/// This the main class of the library. It represents a Pushover app and
/// is tied to a unique API token. When constructing the object it is mandatory to pass
/// an `app-token` as well as a `user-token`.
///
/// Here's a simple example, which sends a pushover notification to a specific device of the user.
/// Note that this class uses a fluent API to configure the properties of a notification.
/// The actual action of sending the notification is triggered by [SendMessageAsync](xref:Pushover.PushoverClient#SendMessageAsync).
/// The ´Async´ Suffix in this method indicates that this action has to be waited for by checking for ´NOT _pushoverClient.Busy´ before
/// sending another notification.
///
/// ```sti
/// PROGRAM MAIN
/// VAR
///   _send : BOOL; // boolean, which can be triggered to send a message
///   _pushoverClient : Pushover.PushoverClient('<your_pushover_apptoken>', '<your_pushover_user>'); 
/// END_VAR
/// ```
/// ```std
/// IF _send
/// THEN
///   _send := FALSE;
///   _pushoverClient
///     .SendMessageAsync('Hello World!');
/// END_IF
///
/// _pushoverClient.Cyclic();
/// ```
{attribute 'conditionalshow_all_locals'}
{attribute 'no_explicit_call' := 'This FB is a CLASS and must be accessed using methods and/or properties'}
FUNCTION_BLOCK PushoverClient IMPLEMENTS IPushoverClient
VAR
  _busy : BOOL;
  _error : BOOL;
  _errorMessage : STRING(255);
  
  _response : STRING(255);
  _request : PushoverRequest;
  _server : Tc2_System.ADSRDWRTEX;
END_VAR
VAR CONSTANT
  _defaultHost : STRING := '127.0.0.1.1.1';
  _defaultPort : UINT := 25733;
END_VAR

/// This property can be used to check if the client is ready for sending a notification. If the client is not 
/// ready or an error occurs during sending (e.g. not internet connection, Pushover Twincat Service is not running, ...)
/// the property [Error](xref:Pushover.PushoverClient#Error) returns `true`.
{attribute 'monitoring' := 'call'}
PROPERTY Busy : BOOL
GET
Busy := _busy;
END_GET
SET // PROTECTED
_busy := Busy;

IF _busy
THEN
  _error := FALSE;
END_IF
END_SET
END_PROPERTY

/// Resets all `WithXXX` statements to their default values.
METHOD Clear : IPushoverClient
VAR
  token : STRING;
  user : STRING;
  host : STRING := '127.0.0.1.1.1';
  port : UINT := 25733;  
END_VAR
token := THIS^.Token;
user := THIS^.User;
host := THIS^.Host;
port := THIS^.Port;

Tc2_System.MEMSET(ADR(_request), 0, SIZEOF(_request));
_request.Priority := PushoverPriority.Normal;
_request.Sound := PushoverSound.Pushover;

THIS^.Token := token;
THIS^.User := user;
THIS^.Host := _defaultHost;
THIS^.Port := _defaultPort;

Clear := THIS^;
END_METHOD

/// This method has to be called cyclically and takes care of the communication with the `Pushover Twincat Service`, which is reached 
/// via [Host](xref:Pushover.PushoverClient#Host) and [Port](xref:Pushover.PushoverClient#Port).
/// You can use the properties [Busy](xref:Pushover.PushoverClient#Busy) and [Error](xref:Pushover.PushoverClient#Error) to check weather an
/// operation was successful (`NOT Busy AND NOT Error`) or failed (`Error`), respectively.
METHOD Cyclic
VAR_INST
  errorTrig : Tc2_Standard.R_TRIG;
END_VAR
IF NOT Busy
THEN
  RETURN;
END_IF

_server(IDXOFFS:=0, 
        WRITELEN:=SIZEOF(_request),
        SRCADDR:=ADR(_request),
        DESTADDR:=ADR(_response),
        READLEN:=SIZEOF(_response),
        WRTRD:=TRUE, 
        TMOUT:=T#5S,
        ERR=>,
        BUSY=>,
        ERRID=>);
  
IF _server.ERR // fallback to proxy
THEN
  Error := TRUE;
  _errorMessage := _response;
ELSIF NOT _server.BUSY 
THEN
  Busy := FALSE;
END_IF
END_METHOD

/// Enables Monospace in the pushover message
/// Either [HTML](xref:Pushover.PushoverClient#EnableHtml) or [Monospace](xref:Pushover.PushoverClient#EnableMonspace) can be enabled
METHOD EnableHtml : IPushoverClient
_request.MessageType := PushoverMessageType.Html;

EnableHtml := THIS^;
END_METHOD

/// Enables HTML in the pushover message
/// Either [HTML](xref:Pushover.PushoverClient#EnableHtml) or [Monospace](xref:Pushover.PushoverClient#EnableMonspace) can be enabled
METHOD EnableMonospace : IPushoverClient
_request.MessageType := PushoverMessageType.Monospace;

EnableMonospace := THIS^;
END_METHOD

/// Returns `true` if any error occured when calling an `XXX_Async` method of this object. The details of the error
/// are available by checking the proeprty
{attribute 'monitoring' := 'call'}
PROPERTY Error : BOOL
GET
Error := _error;
END_GET
SET // PROTECTED
_error := Error;

IF _error
THEN
  _busy := FALSE;
END_IF
END_SET
END_PROPERTY

/// Only valid if `Error=TRUE`, returns the explanation why the call of an `XXX_Async` method failed.
METHOD ErrorMessage : STRING(255);
ErrorMessage := _errorMessage;
END_METHOD

METHOD FB_init : BOOL
VAR_INPUT
	bInitRetains : BOOL; // if TRUE, the retain variables are initialized (warm start / cold start)
	bInCopyCode : BOOL;  // if TRUE, the instance afterwards gets moved into the copy code (online change)
  
  /// The pushover API token
  token : STRING;
  
  /// The user/group key (not e-mail address) of your user (or you),
  /// viewable when logged into the [pushover dashboard](https://pushover.net/login)
  user : STRING;
END_VAR
THIS^.Token := token;
THIS^.User := user;
THIS^.Host := _defaultHost;
THIS^.Port := _defaultPort;

Clear();
END_METHOD

/// Returns the AMS Net Id of the `Pushover Twincat Service`. Defauls to localhost
PROPERTY Host : STRING
GET
Host := _server.NETID;
END_GET
SET
_server(WRTRD := FALSE,
       NETID := Host,
       BUSY=>,
       ERR=>,
       ERRID=>);
END_SET
END_PROPERTY

PROPERTY Port : UINT
GET
Port := _server.PORT;
END_GET
SET
_server(WRTRD := FALSE,
       PORT := Port,
       BUSY=>,
       ERR=>,
       ERRID=>);
END_SET
END_PROPERTY

METHOD SendMessageAsync
VAR_IN_OUT CONSTANT
  title : STRING(255);
  message : STRING(255);
END_VAR
IF NOT Busy
THEN
  _request.TitleLength := Tc2_Standard.LEN(title);
  _request.Title := title;
  _request.MessageLength := Tc2_Standard.LEN(message);
  _request.Message := message;
  
  _server(WRTRD := FALSE,
         IDXGRP:=0,
         BUSY=>,
         ERR=>,
         ERRID=>);    
  Busy := TRUE;
ELSE
  Error := TRUE;
  _errorMessage := 'Client can not executed parallel requests!';
END_IF
END_METHOD

PROPERTY Token : STRING
GET
Token := _request.Token;
END_GET
SET
_request.Token := Token;
_request.TokenLength := Tc2_Standard.LEN(_request.Token);
END_SET
END_PROPERTY

PROPERTY User : STRING
GET
User := _request.User;
END_GET
SET
_request.User := User;
_request.UserLength := Tc2_Standard.LEN(_request.User);
END_SET
END_PROPERTY

/// Callback parameter may be supplied with a publicly-accessible URL that the
/// pushover servers will send a request to when the user has acknowledged your
/// notification.
/// Only used if priority is set to emergency.
METHOD WithCallback : IPushoverClient
VAR_IN_OUT CONSTANT
  callback : STRING(255);
END_VAR
_request.CallbackLength := Tc2_Standard.LEN(callback);
_request.Callback := callback;

WithCallback := THIS^;
END_METHOD

/// Your user's device name to send the message directly to that device,
/// rather than all of the user's devices
METHOD WithDevice : IPushoverClient
VAR_IN_OUT CONSTANT
  device : STRING(80);
END_VAR
_request.DeviceLength := Tc2_Standard.LEN(device);
_request.Device := device;

WithDevice := THIS^;
END_METHOD

/// Specifies how many seconds your notification will continue to be retried for (every retry seconds).
/// Only required if priority is set to emergency.
METHOD WithExpire : IPushoverClient
VAR_INPUT
  expire : INT;
END_VAR
_request.Expire := expire;

WithExpire := THIS^;
END_METHOD

/// Priority of the message
METHOD WithPriority : IPushoverClient
VAR_INPUT
  priority : PushoverPriority;
END_VAR
_request.Priority := priority;

WithPriority := THIS^;
END_METHOD

/// Adds a ttl to the Pushover message
METHOD WithProxy : IPushoverClient
VAR_IN_OUT CONSTANT
  host : STRING(80);
END_VAR
VAR_INPUT
  port : INT;
END_VAR
_request.ProxyHostLength := Tc2_Standard.LEN(host);
_request.ProxyHost := host;
_request.ProxyPort := port;

WithProxy := THIS^;
END_METHOD

/// Specifies how often (in seconds) the Pushover servers will send the same notification to the user.
/// Only required if priority is set to emergency.
METHOD WithRetry : IPushoverClient
VAR_INPUT
  retry : INT;
END_VAR
_request.Retry := retry;

WithRetry := THIS^;
END_METHOD

/// Priority of the message
METHOD WithSound : IPushoverClient
VAR_INPUT
  sound : PushoverSound;
END_VAR
_request.Sound := sound;

WithSound := THIS^;
END_METHOD

/// A Unix timestamp of your message's date and time to display to the user,
/// rather than the time your message is received by the pushover API
METHOD WithTimestamp : IPushoverClient
VAR_INPUT
  timestamp : INT; //< UNIX Timestamp in seconds
END_VAR
_request.Timestamp := timestamp;

WithTimestamp := THIS^;
END_METHOD

/// Adds a ttl to the Pushover message
METHOD WithTimeToLive : IPushoverClient
VAR_INPUT
  ttl : INT; //< Seconds until this message should be automatically removed from the device. Needs to be positive
END_VAR
_request.TimeToLive := ttl;

WithTimeToLive := THIS^;
END_METHOD

/// A supplementary URL to show with your message
METHOD WithUrl : IPushoverClient
VAR_IN_OUT CONSTANT
  url : STRING(255);
END_VAR
_request.UrlLength := Tc2_Standard.LEN(url);
_request.Url := url;

WithUrl := THIS^;
END_METHOD

/// A title for your supplementary URL, otherwise just the URL is shown
METHOD WithUrlTitle : IPushoverClient
VAR_IN_OUT CONSTANT
  urlTitle : STRING(255);
END_VAR
_request.UrlTitleLength := Tc2_Standard.LEN(urlTitle);
_request.UrlTitle := urlTitle;

WithUrlTitle := THIS^;
END_METHOD

END_FUNCTION_BLOCK

(* stored: Version 1.1.0.1, ProductVersion 3.1.4024.12
   POU PushoverClient: Id {7e1e9724-26e2-0084-1004-42ca9b5de5a8}, SpecialFunc None
   Property Busy: Id {72c62e30-e885-4eb2-98b1-f1d26e618bab}
   Get Get: Id {638df4c4-ce17-46ec-9ad7-929d45026307}
   Set Set: Id {72c23c85-7457-4c77-954b-13dc2bbf6698}
   Method Clear: Id {0f0aec67-27b6-49f3-bec9-7f030e47c04d}
   Method Cyclic: Id {426e1ace-8aa7-0373-078f-f6c08bda3162}
   Method EnableHtml: Id {89eb8acd-b285-4eec-86d7-00035e5cd1dd}
   Method EnableMonospace: Id {c310f4b2-c2e7-4a9c-91ed-7d2738403dad}
   Property Error: Id {e66821e4-2ee0-4372-9ea9-1eb4dd33a529}
   Get Get: Id {e7a38956-1dfd-4ffd-92e4-bca9edabac1a}
   Set Set: Id {32d3bb0b-6ab6-467b-877b-dec253655bc9}
   Method ErrorMessage: Id {7b499ef8-eacf-4d4f-8980-fd3275b78050}
   Method FB_init: Id {35c9eeb9-61ee-4ff2-8c41-88a6a762ab87}
   Property Host: Id {d06b2e65-bd92-4aa0-a8cf-123040bf4d63}
   Get Get: Id {a03127e3-650c-4e7b-943a-977d03c8073e}
   Set Set: Id {c8ced228-6a9e-4ba5-b049-2d5511e74bd0}
   Property Port: Id {6d99f1c3-57ba-40cf-a01f-00d80a87bd49}
   Get Get: Id {62cd6a40-8a44-4f9c-bdf5-2065126bdfe3}
   Set Set: Id {e9a96dd4-dec0-4ef1-bb24-acc78eea7c5b}
   Method SendMessageAsync: Id {2514d27a-339b-498f-a48f-770ba2a832fe}
   Property Token: Id {bf5e10e9-5772-4f05-993b-dd3d2d60441b}
   Get Get: Id {d6e8aca1-e3e6-4f04-8a9f-bce9c98cf5a4}
   Set Set: Id {1a083cd8-6ea7-4bd2-9213-fc1474c0c5d4}
   Property User: Id {82b03ea8-9b37-4d8a-bdb9-35faa26390b3}
   Get Get: Id {0226d001-c16a-46fa-ab97-181d7e748daf}
   Set Set: Id {dc42dc15-95ff-482b-b929-6f6f0a82ad3e}
   Method WithCallback: Id {bbf0f02d-aa8b-4a81-b76e-2d539229251b}
   Method WithDevice: Id {8e580a7c-b56f-4317-ad3d-a4179f302058}
   Method WithExpire: Id {0fb39e03-bbfd-4c10-84ee-42256ae2318f}
   Method WithPriority: Id {24bec2e3-b8f2-4b8e-a20b-a7cebcd754b2}
   Method WithProxy: Id {76ef8889-93e9-4000-9e62-e82a5912536b}
   Method WithRetry: Id {dfa2febd-6783-4cf8-9fac-f6f2b50b134c}
   Method WithSound: Id {2f94b457-e6b6-4d90-b02b-1c02343075fc}
   Method WithTimestamp: Id {58dfffc6-9d1f-430f-bf7c-b0b659b98722}
   Method WithTimeToLive: Id {dfa164aa-34bd-4403-ab2b-ee2c20167769}
   Method WithUrl: Id {95ed75c2-d162-4897-889c-2e97e50c34a7}
   Method WithUrlTitle: Id {2fa3cc93-95d4-46b3-830a-74d9f9be2636} *)
